{attribute 'GeneratedUsingTerminal: EK1100-0000-0018'}
{attribute addProperty BoxType "EK1100-0000-0018"}
{attribute addProperty Id "Beckhoff_EK12xxEK1122Beckhoff_EK12xxEK1122_F8B8118B2"}
{attribute addProperty CRC "4034783571"}
{attribute addProperty Size "2"}
{attribute addProperty Name "Beckhoff EK12xx"}
TYPE Beckhoff_EK12xx_F07DE953 EXTENDS EK1100_1FC0878B :
STRUCT
	{attribute addProperty Name "Beckhoff EK12xxEK1122"}
	{attribute addProperty PreviousPort "Beckhoff EK12xx : B"}
	Beckhoff_EK12xxEK1122 : Beckhoff_EK12xxEK1122_F8B8118B;
END_STRUCT
END_TYPE

(* stored: Version 1.2.0.0, ProductVersion 3.1.4024.11
   DUT Beckhoff_EK12xx_F07DE953: Id {8927b9dc-9f3f-452e-9c20-f2b8838ea345} *)
